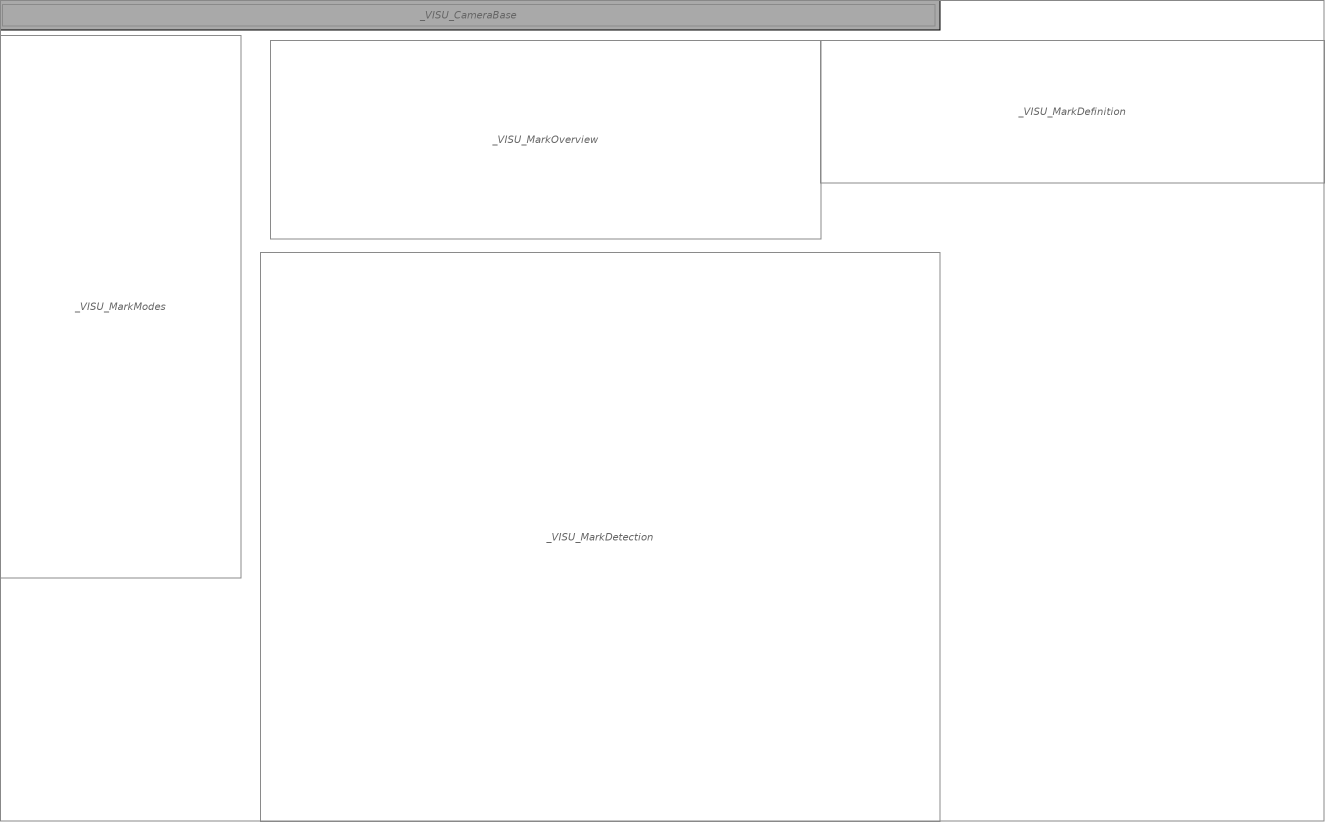
VISUALIZATION _VISU_MarkCamera_WEU  // 1325x822
VAR_IN_OUT
  mInst : FB_MarkCamera_WEU;
END_VAR
    RoundedRectangle (0,0 940x30)
    Frame (270,40 551x199)
        shows _VISU_MarkOverview(mInst := mInst)
    Frame (2,4 933x22)
        shows _VISU_CameraBase(m_Inst := mInst)
    Frame (0,35 241x543)
        shows _VISU_MarkModes(mInst := mInst)
    Frame (260,252 680x570)
        shows _VISU_MarkDetection(mInst := mInst.fbMarkDetection)
    Frame (820,40 505x143)
        shows _VISU_MarkDefinition(mInst := mInst.fbMarkDefinition)
END_VISUALIZATION

(* stored: Version 1.1.0.1, ProductVersion 3.1.4024.11
   Visu _VISU_MarkCamera_WEU: Id {daf9130b-ea3a-4d24-bb53-8b3f847e2ec5} *)
